// TIA Portal V18 export
// export: Created 2026-03-12T16:04:35.9791037Z, ExportSetting WithDefaults, DisplayName Totally Integrated Automation Portal, DisplayVersion V18 Update 5, DisplayName TIA Portal Openness, DisplayVersion V18 Update 5, DisplayName TIA Portal Version Control Interface, DisplayVersion V18, DisplayName SINAMICS Startdrive Advanced, DisplayVersion V18, DisplayName SINAMICS Startdrive G130, G150, S120, S150, SINAMICS MV, S210, DisplayVersion V18, DisplayName SINAMICS Startdrive G110M, G120, G120C, G120D, G120P, G115D, DisplayVersion V18, DisplayName STEP 7 Professional, DisplayVersion V18 Update 5, DisplayName STEP 7 Safety, DisplayVersion V18, DisplayName WinCC Professional, DisplayVersion V18 Update 5
FUNCTION_BLOCK "FB_MOVE_SKID_DECANTADOR_SECUNDARIO"   // FB36, LAD
{ S7_Optimized_Access := 'TRUE' }
VERSION : 0.1
// stored: AutoNumber true, IsIECCheckEnabled false, IsRetainMemResEnabled false, MemoryReserve 100, SetENOAutomatically false, UDAEnableTagReadback false
   VAR_INPUT
      READ_STRUCT_1 : Array[0..10] of Word;
      READ_STRUCT_2 : Array[0..10] of Word;
      READ_STRUCT_3 : Array[0..10] of Word;
   END_VAR
   VAR_OUTPUT
      SKID_1 : Struct
         Falta_Fase : Bool;
         Disjuntor_Motor : Bool;
         Partida_Ponte : Bool;
         Parada_Ponte : Bool;
         Modo_Op : Bool;
         Emergencia : Bool;
         Falha_Inversor : Bool;
      END_STRUCT;
      SKID_2 : Struct
         Falta_Fase : Bool;
         Disjuntor_Motor : Bool;
         Partida_Ponte : Bool;
         Parada_Ponte : Bool;
         Modo_Op : Bool;
         Emergencia : Bool;
         Falha_Inversor : Bool;
      END_STRUCT;
      SKID_3 : Struct
         Falta_Fase : Bool;
         Disjuntor_Motor : Bool;
         Partida_Ponte : Bool;
         Parada_Ponte : Bool;
         Modo_Op : Bool;
         Emergencia : Bool;
         Falha_Inversor : Bool;
      END_STRUCT;
   END_VAR
   VAR_IN_OUT
      MOTOR_1 : "MotorDados";
      MOTOR_2 : "MotorDados";
      MOTOR_3 : "MotorDados";
   END_VAR
   VAR_TEMP   // added for the SCL form of the ladder/FBD networks
      _w1 : Bool;
   END_VAR
BEGIN

REGION Network 1: MOVE_SKID_1
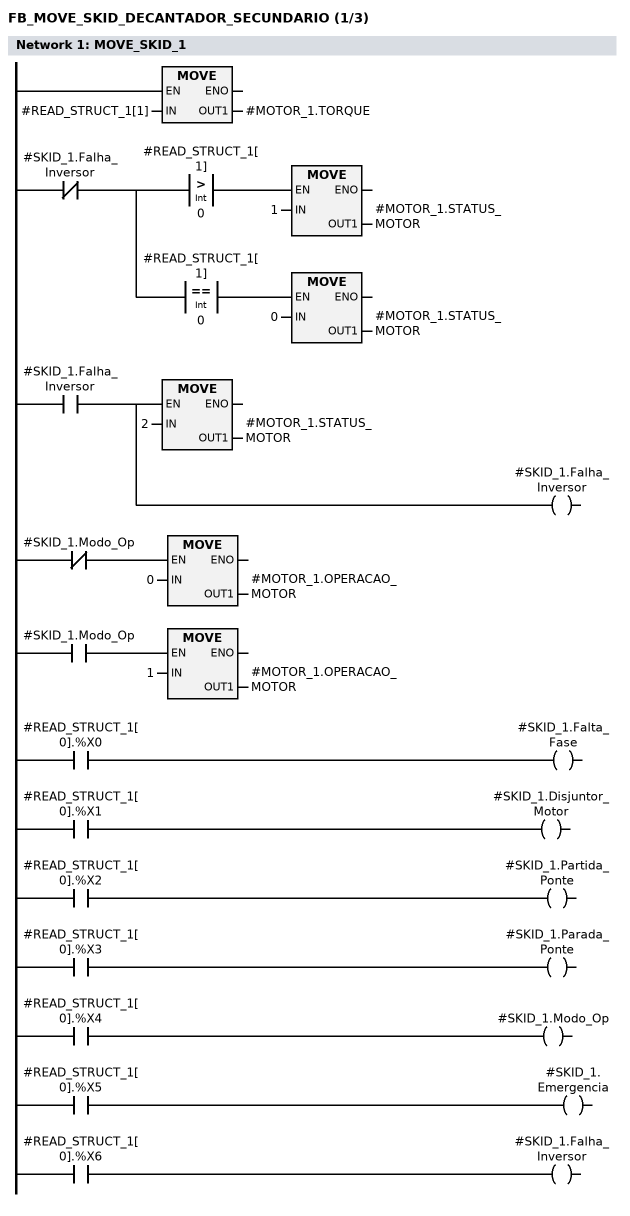
   RUNG wire#powerrail
      Move(in := #READ_STRUCT_1[1], out1 => #MOTOR_1.TORQUE)
   END_RUNG
   RUNG wire#powerrail
      I_Contact( #SKID_1.Falha_Inversor )
      wire#w1
      { S7_Templates := "SrcType := Int" } GT_Contact(in1 := #READ_STRUCT_1[1], in2 := 0)
      Move(in := 1, out1 => #MOTOR_1.STATUS_MOTOR)
   END_RUNG
   RUNG wire#w1
      { S7_Templates := "SrcType := Int" } EQ_Contact(in1 := #READ_STRUCT_1[1], in2 := 0)
      Move(in := 0, out1 => #MOTOR_1.STATUS_MOTOR)
   END_RUNG
   RUNG wire#powerrail
      Contact( #SKID_1.Falha_Inversor )
      wire#w2
      Move(in := 2, out1 => #MOTOR_1.STATUS_MOTOR)
   END_RUNG
   RUNG wire#w2
      Coil( #SKID_1.Falha_Inversor )
   END_RUNG
   RUNG wire#powerrail
      I_Contact( #SKID_1.Modo_Op )
      Move(in := 0, out1 => #MOTOR_1.OPERACAO_MOTOR)
   END_RUNG
   RUNG wire#powerrail
      Contact( #SKID_1.Modo_Op )
      Move(in := 1, out1 => #MOTOR_1.OPERACAO_MOTOR)
   END_RUNG
   RUNG wire#powerrail
      Contact( #READ_STRUCT_1[0].%X0 )
      Coil( #SKID_1.Falta_Fase )
   END_RUNG
   RUNG wire#powerrail
      Contact( #READ_STRUCT_1[0].%X1 )
      Coil( #SKID_1.Disjuntor_Motor )
   END_RUNG
   RUNG wire#powerrail
      Contact( #READ_STRUCT_1[0].%X2 )
      Coil( #SKID_1.Partida_Ponte )
   END_RUNG
   RUNG wire#powerrail
      Contact( #READ_STRUCT_1[0].%X3 )
      Coil( #SKID_1.Parada_Ponte )
   END_RUNG
   RUNG wire#powerrail
      Contact( #READ_STRUCT_1[0].%X4 )
      Coil( #SKID_1.Modo_Op )
   END_RUNG
   RUNG wire#powerrail
      Contact( #READ_STRUCT_1[0].%X5 )
      Coil( #SKID_1.Emergencia )
   END_RUNG
   RUNG wire#powerrail
      Contact( #READ_STRUCT_1[0].%X6 )
      Coil( #SKID_1.Falha_Inversor )
   END_RUNG
   // the same network as SCL:
   #MOTOR_1.TORQUE := #READ_STRUCT_1[1];
   #_w1 := NOT #SKID_1.Falha_Inversor;
   IF #_w1 AND (#READ_STRUCT_1[1] > 0) THEN #MOTOR_1.STATUS_MOTOR := 1; END_IF;
   IF #_w1 AND (#READ_STRUCT_1[1] = 0) THEN #MOTOR_1.STATUS_MOTOR := 0; END_IF;
   IF #SKID_1.Falha_Inversor THEN #MOTOR_1.STATUS_MOTOR := 2; END_IF;
   #SKID_1.Falha_Inversor := #SKID_1.Falha_Inversor;
   IF NOT #SKID_1.Modo_Op THEN #MOTOR_1.OPERACAO_MOTOR := 0; END_IF;
   IF #SKID_1.Modo_Op THEN #MOTOR_1.OPERACAO_MOTOR := 1; END_IF;
   #SKID_1.Falta_Fase := #READ_STRUCT_1[0].%X0;
   #SKID_1.Disjuntor_Motor := #READ_STRUCT_1[0].%X1;
   #SKID_1.Partida_Ponte := #READ_STRUCT_1[0].%X2;
   #SKID_1.Parada_Ponte := #READ_STRUCT_1[0].%X3;
   #SKID_1.Modo_Op := #READ_STRUCT_1[0].%X4;
   #SKID_1.Emergencia := #READ_STRUCT_1[0].%X5;
   #SKID_1.Falha_Inversor := #READ_STRUCT_1[0].%X6;
END_REGION

REGION Network 2: MOVE_SKID_2
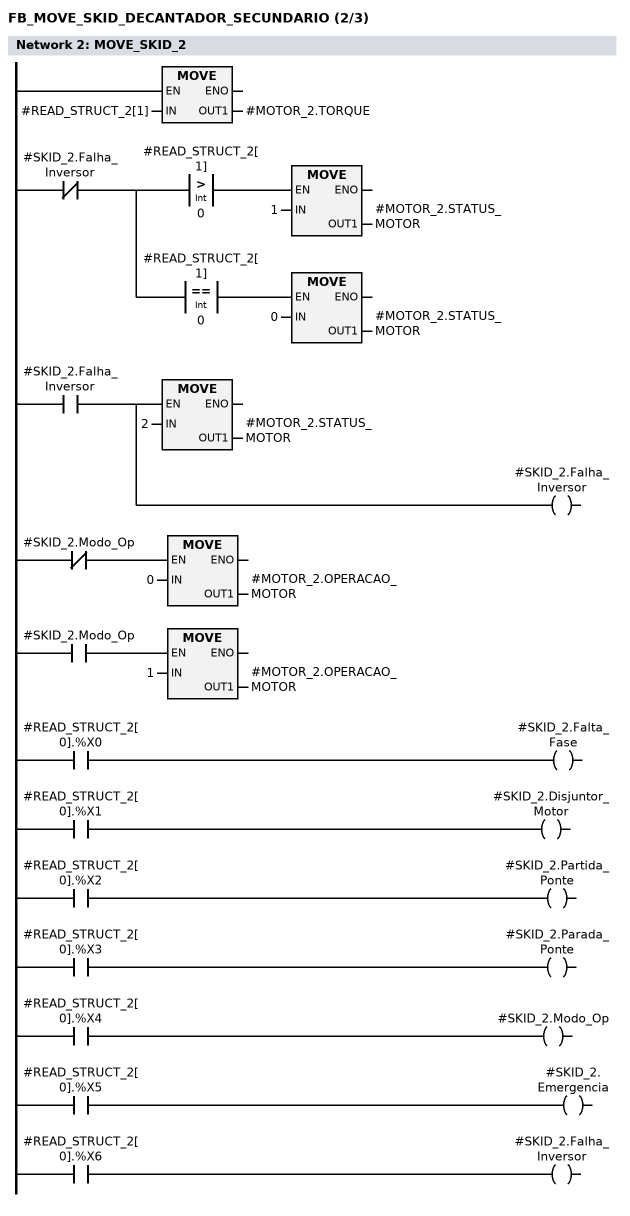
   RUNG wire#powerrail
      Move(in := #READ_STRUCT_2[1], out1 => #MOTOR_2.TORQUE)
   END_RUNG
   RUNG wire#powerrail
      I_Contact( #SKID_2.Falha_Inversor )
      wire#w1
      { S7_Templates := "SrcType := Int" } GT_Contact(in1 := #READ_STRUCT_2[1], in2 := 0)
      Move(in := 1, out1 => #MOTOR_2.STATUS_MOTOR)
   END_RUNG
   RUNG wire#w1
      { S7_Templates := "SrcType := Int" } EQ_Contact(in1 := #READ_STRUCT_2[1], in2 := 0)
      Move(in := 0, out1 => #MOTOR_2.STATUS_MOTOR)
   END_RUNG
   RUNG wire#powerrail
      Contact( #SKID_2.Falha_Inversor )
      wire#w2
      Move(in := 2, out1 => #MOTOR_2.STATUS_MOTOR)
   END_RUNG
   RUNG wire#w2
      Coil( #SKID_2.Falha_Inversor )
   END_RUNG
   RUNG wire#powerrail
      I_Contact( #SKID_2.Modo_Op )
      Move(in := 0, out1 => #MOTOR_2.OPERACAO_MOTOR)
   END_RUNG
   RUNG wire#powerrail
      Contact( #SKID_2.Modo_Op )
      Move(in := 1, out1 => #MOTOR_2.OPERACAO_MOTOR)
   END_RUNG
   RUNG wire#powerrail
      Contact( #READ_STRUCT_2[0].%X0 )
      Coil( #SKID_2.Falta_Fase )
   END_RUNG
   RUNG wire#powerrail
      Contact( #READ_STRUCT_2[0].%X1 )
      Coil( #SKID_2.Disjuntor_Motor )
   END_RUNG
   RUNG wire#powerrail
      Contact( #READ_STRUCT_2[0].%X2 )
      Coil( #SKID_2.Partida_Ponte )
   END_RUNG
   RUNG wire#powerrail
      Contact( #READ_STRUCT_2[0].%X3 )
      Coil( #SKID_2.Parada_Ponte )
   END_RUNG
   RUNG wire#powerrail
      Contact( #READ_STRUCT_2[0].%X4 )
      Coil( #SKID_2.Modo_Op )
   END_RUNG
   RUNG wire#powerrail
      Contact( #READ_STRUCT_2[0].%X5 )
      Coil( #SKID_2.Emergencia )
   END_RUNG
   RUNG wire#powerrail
      Contact( #READ_STRUCT_2[0].%X6 )
      Coil( #SKID_2.Falha_Inversor )
   END_RUNG
   // the same network as SCL:
   #MOTOR_2.TORQUE := #READ_STRUCT_2[1];
   #_w1 := NOT #SKID_2.Falha_Inversor;
   IF #_w1 AND (#READ_STRUCT_2[1] > 0) THEN #MOTOR_2.STATUS_MOTOR := 1; END_IF;
   IF #_w1 AND (#READ_STRUCT_2[1] = 0) THEN #MOTOR_2.STATUS_MOTOR := 0; END_IF;
   IF #SKID_2.Falha_Inversor THEN #MOTOR_2.STATUS_MOTOR := 2; END_IF;
   #SKID_2.Falha_Inversor := #SKID_2.Falha_Inversor;
   IF NOT #SKID_2.Modo_Op THEN #MOTOR_2.OPERACAO_MOTOR := 0; END_IF;
   IF #SKID_2.Modo_Op THEN #MOTOR_2.OPERACAO_MOTOR := 1; END_IF;
   #SKID_2.Falta_Fase := #READ_STRUCT_2[0].%X0;
   #SKID_2.Disjuntor_Motor := #READ_STRUCT_2[0].%X1;
   #SKID_2.Partida_Ponte := #READ_STRUCT_2[0].%X2;
   #SKID_2.Parada_Ponte := #READ_STRUCT_2[0].%X3;
   #SKID_2.Modo_Op := #READ_STRUCT_2[0].%X4;
   #SKID_2.Emergencia := #READ_STRUCT_2[0].%X5;
   #SKID_2.Falha_Inversor := #READ_STRUCT_2[0].%X6;
END_REGION

REGION Network 3: MOVE_SKID_3
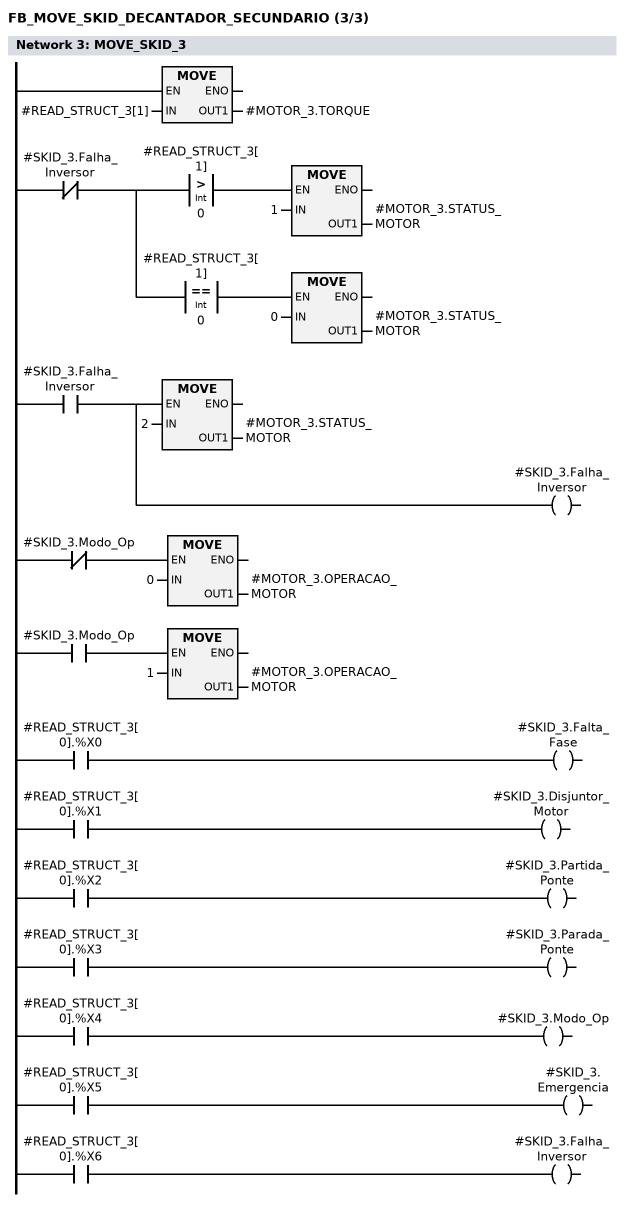
   RUNG wire#powerrail
      Move(in := #READ_STRUCT_3[1], out1 => #MOTOR_3.TORQUE)
   END_RUNG
   RUNG wire#powerrail
      I_Contact( #SKID_3.Falha_Inversor )
      wire#w1
      { S7_Templates := "SrcType := Int" } GT_Contact(in1 := #READ_STRUCT_3[1], in2 := 0)
      Move(in := 1, out1 => #MOTOR_3.STATUS_MOTOR)
   END_RUNG
   RUNG wire#w1
      { S7_Templates := "SrcType := Int" } EQ_Contact(in1 := #READ_STRUCT_3[1], in2 := 0)
      Move(in := 0, out1 => #MOTOR_3.STATUS_MOTOR)
   END_RUNG
   RUNG wire#powerrail
      Contact( #SKID_3.Falha_Inversor )
      wire#w2
      Move(in := 2, out1 => #MOTOR_3.STATUS_MOTOR)
   END_RUNG
   RUNG wire#w2
      Coil( #SKID_3.Falha_Inversor )
   END_RUNG
   RUNG wire#powerrail
      I_Contact( #SKID_3.Modo_Op )
      Move(in := 0, out1 => #MOTOR_3.OPERACAO_MOTOR)
   END_RUNG
   RUNG wire#powerrail
      Contact( #SKID_3.Modo_Op )
      Move(in := 1, out1 => #MOTOR_3.OPERACAO_MOTOR)
   END_RUNG
   RUNG wire#powerrail
      Contact( #READ_STRUCT_3[0].%X0 )
      Coil( #SKID_3.Falta_Fase )
   END_RUNG
   RUNG wire#powerrail
      Contact( #READ_STRUCT_3[0].%X1 )
      Coil( #SKID_3.Disjuntor_Motor )
   END_RUNG
   RUNG wire#powerrail
      Contact( #READ_STRUCT_3[0].%X2 )
      Coil( #SKID_3.Partida_Ponte )
   END_RUNG
   RUNG wire#powerrail
      Contact( #READ_STRUCT_3[0].%X3 )
      Coil( #SKID_3.Parada_Ponte )
   END_RUNG
   RUNG wire#powerrail
      Contact( #READ_STRUCT_3[0].%X4 )
      Coil( #SKID_3.Modo_Op )
   END_RUNG
   RUNG wire#powerrail
      Contact( #READ_STRUCT_3[0].%X5 )
      Coil( #SKID_3.Emergencia )
   END_RUNG
   RUNG wire#powerrail
      Contact( #READ_STRUCT_3[0].%X6 )
      Coil( #SKID_3.Falha_Inversor )
   END_RUNG
   // the same network as SCL:
   #MOTOR_3.TORQUE := #READ_STRUCT_3[1];
   #_w1 := NOT #SKID_3.Falha_Inversor;
   IF #_w1 AND (#READ_STRUCT_3[1] > 0) THEN #MOTOR_3.STATUS_MOTOR := 1; END_IF;
   IF #_w1 AND (#READ_STRUCT_3[1] = 0) THEN #MOTOR_3.STATUS_MOTOR := 0; END_IF;
   IF #SKID_3.Falha_Inversor THEN #MOTOR_3.STATUS_MOTOR := 2; END_IF;
   #SKID_3.Falha_Inversor := #SKID_3.Falha_Inversor;
   IF NOT #SKID_3.Modo_Op THEN #MOTOR_3.OPERACAO_MOTOR := 0; END_IF;
   IF #SKID_3.Modo_Op THEN #MOTOR_3.OPERACAO_MOTOR := 1; END_IF;
   #SKID_3.Falta_Fase := #READ_STRUCT_3[0].%X0;
   #SKID_3.Disjuntor_Motor := #READ_STRUCT_3[0].%X1;
   #SKID_3.Partida_Ponte := #READ_STRUCT_3[0].%X2;
   #SKID_3.Parada_Ponte := #READ_STRUCT_3[0].%X3;
   #SKID_3.Modo_Op := #READ_STRUCT_3[0].%X4;
   #SKID_3.Emergencia := #READ_STRUCT_3[0].%X5;
   #SKID_3.Falha_Inversor := #READ_STRUCT_3[0].%X6;
END_REGION
END_FUNCTION_BLOCK
